TYPE ST_TsDiagObjectsEL2904 :
(*******************************************************************************************************
Description			:	Index 16#800E Diagnostic objects
Supported terminals : 	EL2904
Documentation 		:	EL2904 TwinSAFE output terminal with 4 fail-safe outputs
Version/Date 		:	V1.6.2/02.10.2015
********************************************************************************************************)
STRUCT
	
	nDummyData1								:ARRAY[0..10] OF UINT;

(* Error at the outputs *)
	nErrorOutputs							:UINT;

(* Supply error *)
	nSupplyError							:UINT;

(* Temperature error *)
	nTemperatureError						:UINT;

	nDummyData2								:ARRAY[0..1] OF UINT;

END_STRUCT
END_TYPE
(* End *)

(* stored: Version 1.1.0.1, ProductVersion 3.1.4022.16
   DUT ST_TsDiagObjectsEL2904: Id {9f174f01-b5fb-43fe-9b79-943f15fdd351} *)
